// TIA Portal V16 export
// export: Created 2022-09-01T14:29:26.6530248Z, ExportSetting WithDefaults, DisplayName Totally Integrated Automation Portal, DisplayVersion V16, DisplayName TIA Portal Version Control Interface, DisplayVersion V16, DisplayName TIA Portal Openness, DisplayVersion V16, DisplayName STEP 7 Professional, DisplayVersion V16, DisplayName STEP 7 Safety, DisplayVersion V16, DisplayName WinCC Advanced, DisplayVersion V16
VAR_GLOBAL   // PLC tag table "Falhas"
   DISPARO_DIF_3Q1_32 AT %I0.0 : Bool;
   DISPARO_DIFERENCIAL_3Q3 AT %I0.1 : Bool;
   DISPARO_DIFERENCIAL_4Q1_4Q2 AT %I0.2 : Bool;
   FALHA_24VDC AT %I0.3 : Bool;
   FALHA_220VAC AT %I0.4 : Bool;
   FALHA_24VAC AT %I0.5 : Bool;
END_VAR
